FUNCTION_BLOCK ActivateTrackForMover IMPLEMENTS ITask
VAR_INPUT
END_VAR
VAR_OUTPUT
END_VAR
VAR
	mcActivateTrack : Tc3_McCollisionAvoidance.MC_ActivateTrack;
	_axis : REFERENCE TO Tc2_MC2.AXIS_REF;
	State: INT;
	_done: BOOL;
	_error: BOOL;
	_busy: BOOL;
	_ActivateTrack : BOOL;
	_newTrackId : OTCID;
END_VAR

CASE State OF
	0:
		IF _ActivateTrack THEN
			_done := FALSE;
			_error := FALSE;
			_busy := TRUE;
			mcActivateTrack.Execute := TRUE;
			IF mcActivateTrack.Busy THEN
				State := 10;
				_ActivateTrack := FALSE;
			END_IF
		END_IF
	
	10:
		IF NOT mcActivateTrack.Busy THEN
			IF mcActivateTrack.Done THEN
				_done := TRUE;
				_newTrackId := mcActivateTrack.TrackId;
			ELSIF mcActivateTrack.Error THEN
				_error := TRUE;
			END_IF
			_busy := FALSE;
			mcActivateTrack.Execute := FALSE;
			State := 0;
		END_IF
END_CASE

mcActivateTrack(Axis := _axis);

{warning 'add method implementation '}
METHOD Abort : BOOL
mcActivateTrack.Execute := FALSE;
_busy := FALSE;
_ActivateTrack := FALSE;
Abort := TRUE;
State := 0;
END_METHOD

{warning 'add property implementation'}
PROPERTY Busy : BOOL
GET
Busy := _busy;
END_GET
END_PROPERTY

{warning 'add property implementation'}
PROPERTY Done : BOOL
GET
Done := _done;
END_GET
END_PROPERTY

{warning 'add property implementation'}
PROPERTY Error : BOOL
GET
Error := _error;
END_GET
END_PROPERTY

METHOD PUBLIC Execute : BOOL
VAR_INPUT
	Track : OTCID;
END_VAR
Execute := _ActivateTrack := TRUE;
mcActivateTrack.TrackId := Track;
END_METHOD

METHOD FB_init : BOOL
VAR_INPUT
	bInitRetains : BOOL; // if TRUE, the retain variables are initialized (warm start / cold start)
	bInCopyCode : BOOL;  // if TRUE, the instance afterwards gets moved into the copy code (online change)
	axis : reference TO AXIS_REF;
END_VAR
_axis REF= axis;
END_METHOD

PROPERTY PUBLIC NewTrackId : OTCID
GET
NewTrackId := _newTrackId;
END_GET
END_PROPERTY

END_FUNCTION_BLOCK

(* stored: Version 1.1.0.1, ProductVersion 3.1.4024.11
   POU ActivateTrackForMover: Id {35e3472a-6554-4314-81dc-6f0a8778c0a3}, SpecialFunc None
   Method Abort: Id {feb92e4a-5af0-464c-bf77-407b1ff76646}
   Property Busy: Id {ba2dc81f-a76e-4b6f-a981-60a2cf3b69aa}
   Get Get: Id {f6a8b8bb-a66d-46ae-9807-89fa205ab02d}
   Property Done: Id {c1a82c72-356d-44af-9a2d-d30258c82752}
   Get Get: Id {8cbf4d9c-de32-4a6d-b644-3c51b27ace4f}
   Property Error: Id {4f8688ec-7f9e-4273-a9cd-cdb8dfc358a0}
   Get Get: Id {30faecb5-a98b-47f8-b354-59f7ea76abb6}
   Method Execute: Id {5bda0256-96a6-4784-813e-6a9b4c7cbfd1}
   Method FB_init: Id {3a4ead5e-4416-43d1-b710-bb1444054ab9}
   Property NewTrackId: Id {81e55462-ab9a-4701-8b1c-501e85b6459e}
   Get Get: Id {34911b80-2212-4751-995c-4be8cd54a183} *)
